% RSLogix 500 project P3_ABIOLA_A_V22 BRANCHED V2_BAK156.RSS, saved by version 8.30.00.16 %
PROJECT "UNTITLED"    % processor: Bul.1763 MicroLogix 1100 Series B %

PROGRAM FILES
  LAD 2   2 rungs
  LAD 3 "PSEUDO IO"  13 rungs  % Contains all the assigned memery address used  %

DATA FILES
  O0 OUTPUT  4 elements
  I1 INPUT  6 elements
  S2 STATUS  66 elements
  B3 BINARY  1 elements
  T4 TIMER  4 elements
  C5 COUNTER  3 elements
  R6 CONTROL  1 elements
  N7 INTEGER  11 elements
  F8 FLOAT  1 elements
  ST9 STRFRBCSCN  40 elements  % Writes string from bar code scanner to PLC %
  ST10 STRING  10 elements

LADDER 2
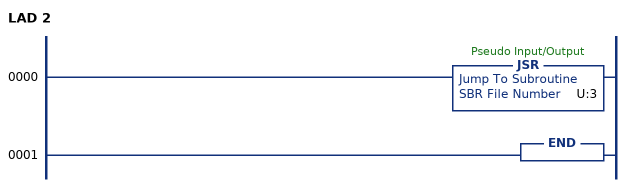
% Rung: 0 %
SOR JSR U:3 EOR
%   U:3  "Pseudo Input/Output" %
% Rung: 1 %
SOR END EOR

LADDER 3 "PSEUDO IO"    % Contains all the assigned memery address used  %
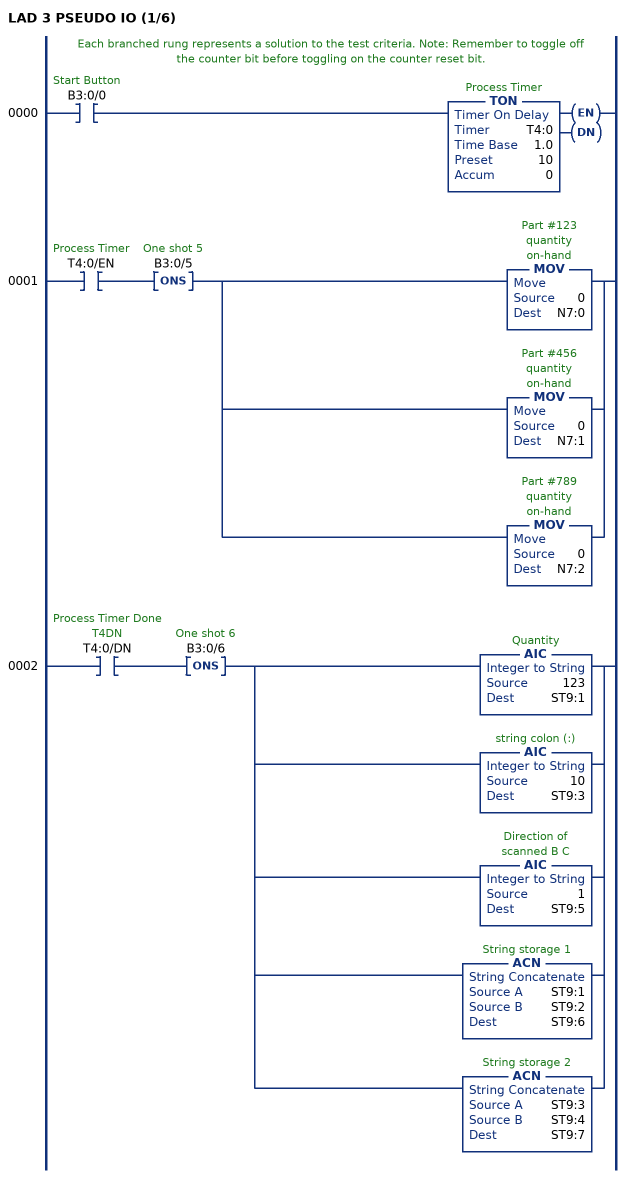
% Rung: 0 %
% Each branched rung represents a solution to the test criteria. Note: Remember to toggle off the counter bit before toggling on the counter reset bit. %
SOR XIC B3:0/0 TON T4:0 1.0 10 0 EOR
%   B3:0/0  "Start Button" %
%   T4:0  "Process Timer" %
% Rung: 1 %
SOR XIC T4:0/EN ONS B3:0/5 BST MOV 0 N7:0 NXB BST MOV 0 N7:1 NXB MOV 0 N7:2 BND BND EOR
%   T4:0  "Process Timer" %
%   B3:0/5  "One shot 5" %
%   N7:0  "Part #123 quantity on-hand" %
%   N7:1  "Part #456 quantity on-hand" %
%   N7:2  "Part #789 quantity on-hand" %
% Rung: 2 %
SOR XIC T4:0/DN ONS B3:0/6 BST AIC 123 ST9:1 NXB BST AIC 10 ST9:3 NXB BST AIC 1 ST9:5 NXB BST ACN ST9:1 ST9:2 ST9:6 NXB ACN ST9:3 ST9:4 ST9:7 BND BND BND BND EOR
%   T4:0/DN  T4DN  "Process Timer Done" %
%   B3:0/6  "One shot 6" %
%   ST9:1  "Quantity" %
%   ST9:3  "string colon (:)" %
%   ST9:5  "Direction of scanned B C" %
%   ST9:2  "String Quantity from Bar-code scanner" %
%   ST9:6  "String storage 1" %
%   ST9:4  "Concatination of colon (:) with direction from BCS" %
%   ST9:7  "String storage 2" %

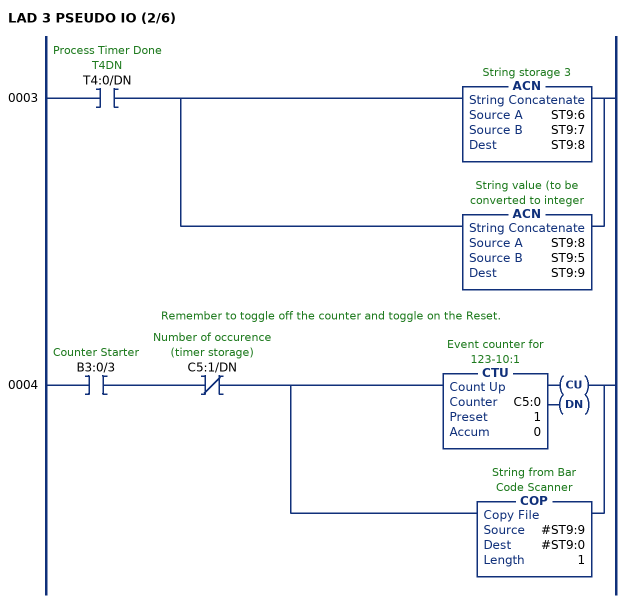
% Rung: 3 %
SOR XIC T4:0/DN BST ACN ST9:6 ST9:7 ST9:8 NXB ACN ST9:8 ST9:5 ST9:9 BND EOR
%   T4:0/DN  T4DN  "Process Timer Done" %
%   ST9:6  "String storage 1" %
%   ST9:7  "String storage 2" %
%   ST9:8  "String storage 3" %
%   ST9:5  "Direction of scanned B C" %
%   ST9:9  "String value (to be converted to integer" %
% Rung: 4 %
% Remember to toggle off the counter and toggle on the Reset. %
SOR XIC B3:0/3 XIO C5:1/DN BST CTU C5:0 1 0 NXB COP #ST9:9 #ST9:0 1 BND EOR
%   B3:0/3  "Counter Starter" %
%   C5:1/DN  "Number of occurence (timer storage)" %
%   C5:0  "Event counter for 123-10:1" %
%   ST9:9  "String value (to be converted to integer" %
%   ST9:0  "String from Bar Code Scanner" %

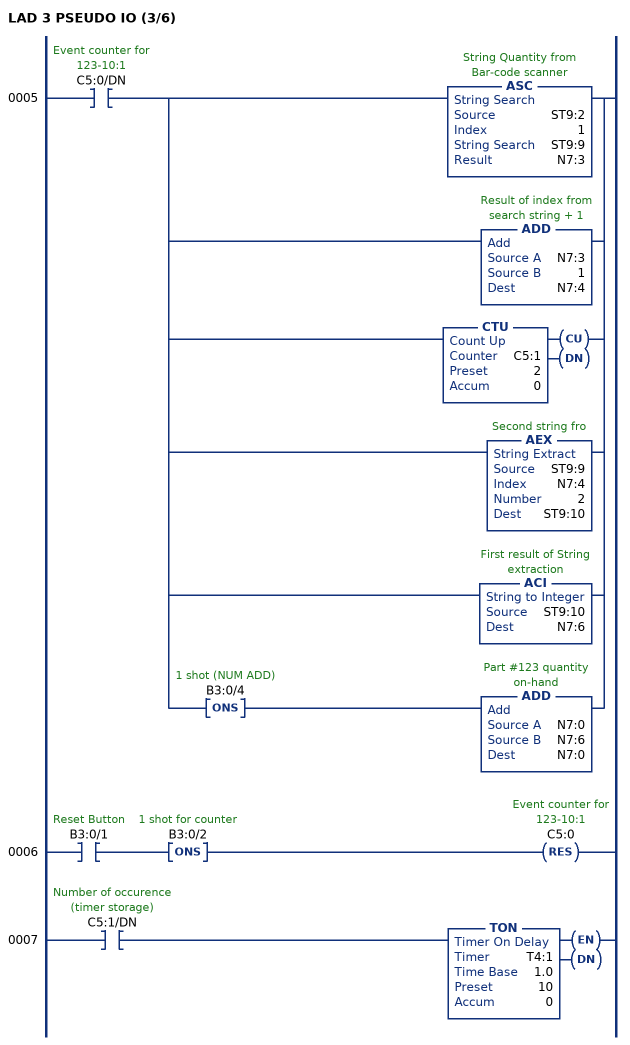
% Rung: 5 %
SOR XIC C5:0/DN BST BST ASC ST9:2 1 ST9:9 N7:3 NXB BST ADD N7:3 1 N7:4 NXB CTU C5:1 2 0 BND BND NXB BST AEX ST9:9 N7:4 2 ST9:10 NXB BST ACI ST9:10 N7:6 NXB ONS B3:0/4 ADD N7:0 N7:6 N7:0 BND BND BND EOR
%   C5:0  "Event counter for 123-10:1" %
%   ST9:2  "String Quantity from Bar-code scanner" %
%   ST9:9  "String value (to be converted to integer" %
%   N7:3  "Constant value of 10" %
%   N7:4  "Result of index from search string + 1" %
%   ST9:10  "Second string fro" %
%   N7:6  "First result of String extraction" %
%   B3:0/4  "1 shot (NUM ADD)" %
%   N7:0  "Part #123 quantity on-hand" %
% Rung: 6 %
SOR XIC B3:0/1 ONS B3:0/2 RES C5:0 EOR
%   B3:0/1  "Reset Button" %
%   B3:0/2  "1 shot for counter" %
%   C5:0  "Event counter for 123-10:1" %
% Rung: 7 %
SOR XIC C5:1/DN TON T4:1 1.0 10 0 EOR
%   C5:1/DN  "Number of occurence (timer storage)" %

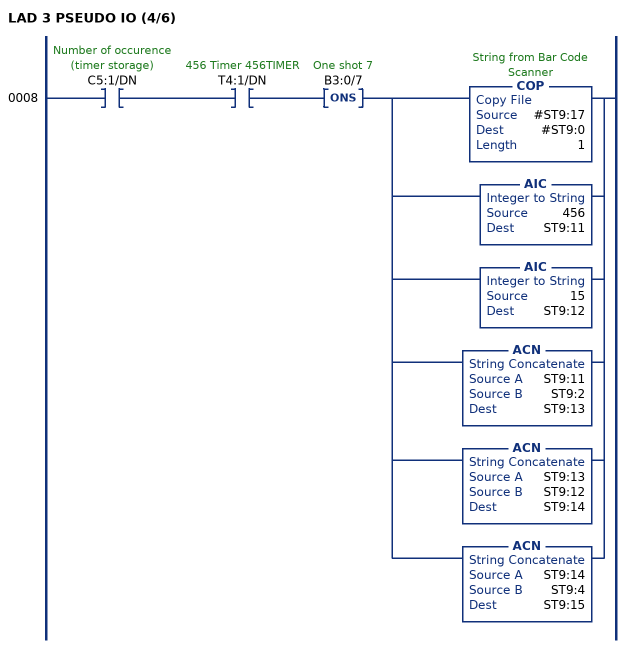
% Rung: 8 %
SOR XIC C5:1/DN XIC T4:1/DN ONS B3:0/7 BST BST COP #ST9:17 #ST9:0 1 NXB AIC 456 ST9:11 BND NXB AIC 15 ST9:12 NXB ACN ST9:11 ST9:2 ST9:13 NXB ACN ST9:13 ST9:12 ST9:14 NXB ACN ST9:14 ST9:4 ST9:15 BND EOR
%   C5:1/DN  "Number of occurence (timer storage)" %
%   T4:1/DN  456TIMER  "456 Timer" %
%   B3:0/7  "One shot 7" %
%   ST9:0  "String from Bar Code Scanner" %
%   ST9:2  "String Quantity from Bar-code scanner" %
%   ST9:4  "Concatination of colon (:) with direction from BCS" %

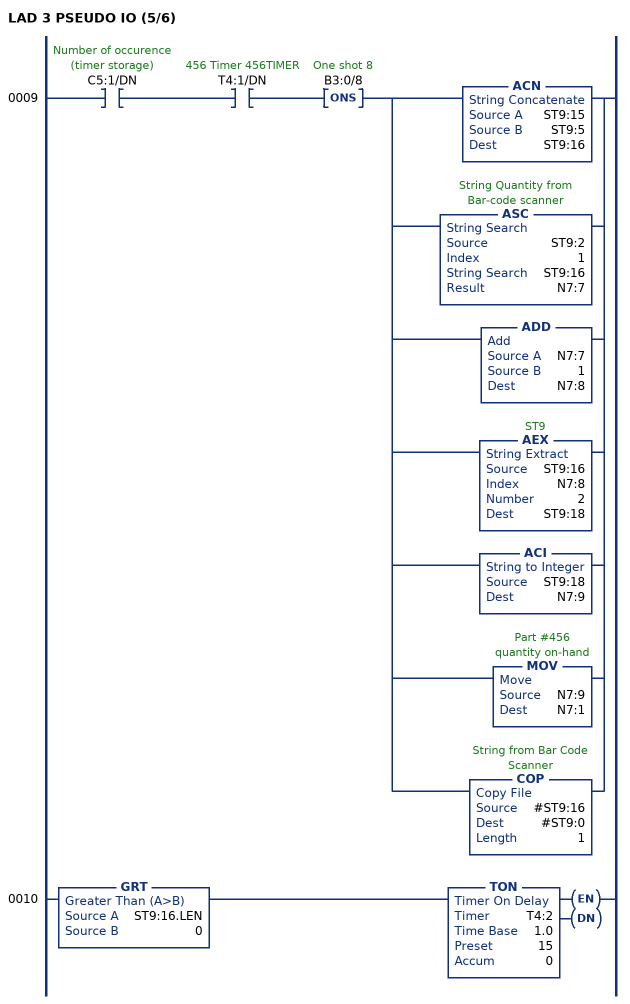
% Rung: 9 %
SOR XIC C5:1/DN XIC T4:1/DN ONS B3:0/8 BST ACN ST9:15 ST9:5 ST9:16 NXB ASC ST9:2 1 ST9:16 N7:7 NXB BST ADD N7:7 1 N7:8 NXB BST BST AEX ST9:16 N7:8 2 ST9:18 NXB ACI ST9:18 N7:9 BND NXB BST MOV N7:9 N7:1 NXB COP #ST9:16 #ST9:0 1 BND BND BND BND EOR
%   C5:1/DN  "Number of occurence (timer storage)" %
%   T4:1/DN  456TIMER  "456 Timer" %
%   B3:0/8  "One shot 8" %
%   ST9:5  "Direction of scanned B C" %
%   ST9:2  "String Quantity from Bar-code scanner" %
%   ST9:18  ST9 %
%   N7:1  "Part #456 quantity on-hand" %
%   ST9:0  "String from Bar Code Scanner" %
% Rung: 10 %
SOR GRT ST9:16.LEN 0 TON T4:2 1.0 15 0 EOR

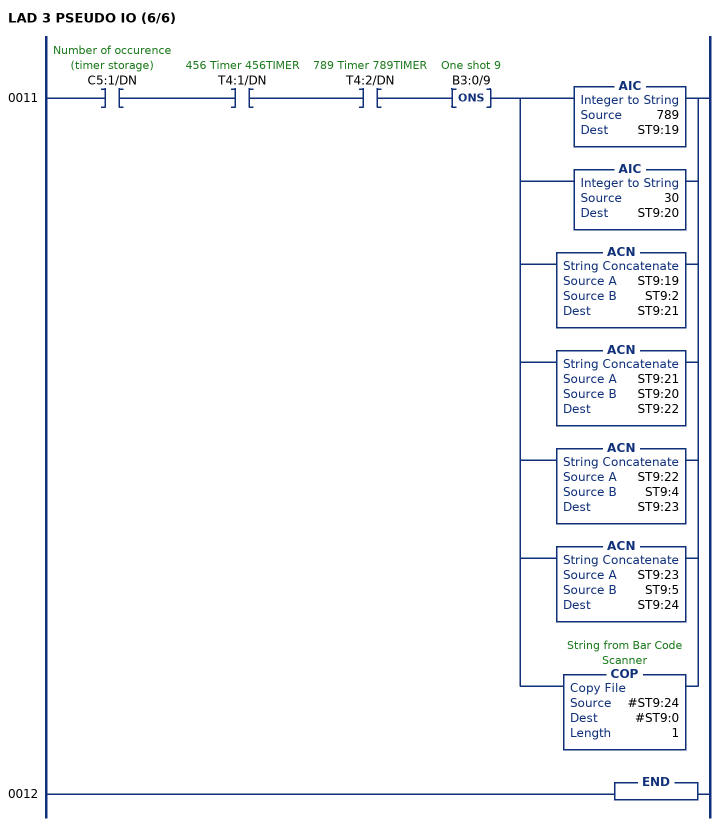
% Rung: 11 %
SOR XIC C5:1/DN XIC T4:1/DN XIC T4:2/DN ONS B3:0/9 BST AIC 789 ST9:19 NXB AIC 30 ST9:20 NXB ACN ST9:19 ST9:2 ST9:21 NXB ACN ST9:21 ST9:20 ST9:22 NXB ACN ST9:22 ST9:4 ST9:23 NXB BST ACN ST9:23 ST9:5 ST9:24 NXB COP #ST9:24 #ST9:0 1 BND BND EOR
%   C5:1/DN  "Number of occurence (timer storage)" %
%   T4:1/DN  456TIMER  "456 Timer" %
%   T4:2/DN  789TIMER  "789 Timer" %
%   B3:0/9  "One shot 9" %
%   ST9:2  "String Quantity from Bar-code scanner" %
%   ST9:4  "Concatination of colon (:) with direction from BCS" %
%   ST9:5  "Direction of scanned B C" %
%   ST9:0  "String from Bar Code Scanner" %
% Rung: 12 %
SOR END EOR

OTHER DOCUMENTED ADDRESSES
  B3:0/10  LN789  "Start line 789-30:1"
  C5:0.ACC  "Number of count storage"
  C5:0/CU  "Process counter"
  C5:2  456COUNTER  "456 Counter"
  C5:2/DN  "LN456 counter"
  N7:5  "String colon (:) converted to integer"
  ST9:2.0  "Result of Constant Multiplication with -1"
  ST10:1.0  "String len"

DATA TABLE (non-zero values as saved)
DATA T4
% .PRE .ACC %
% T4:0 % 10 0
% T4:1 % 10 0
% T4:2 % 15 0
% T4:3 % 10 0
DATA C5
% .PRE .ACC %
% C5:0 % 1 0
% C5:1 % 2 0
% C5:2 % 1 0
DATA ST9
% ST9:2 % "-"
% ST9:4 % ":"
% ST9:17 % " "
